FUNCTION_BLOCK HashMap IMPLEMENTS Map
VAR_INPUT
END_VAR
VAR_OUTPUT
END_VAR
VAR
END_VAR

END_FUNCTION_BLOCK

(* stored: Version 1.1.0.1, ProductVersion 3.1.4024.11
   POU HashMap: Id {034d47c3-248f-4e5a-a7e3-eda5f7ee95dc}, SpecialFunc None *)
